ORGANIZATION_BLOCK "Main"
TITLE = "Main Program Sweep (Cycle)"
{ S7_Optimized_Access := 'TRUE' }
VERSION : 0.1

BEGIN
	"FB_HGU_Motor_Control_Simple_DB"();


END_ORGANIZATION_BLOCK

